// TIA Portal V17 export
// export: Created 2022-08-15T12:48:21.8497446Z, ExportSetting WithDefaults, DisplayName Totally Integrated Automation Portal, DisplayVersion V17, DisplayName TIA Portal Openness, DisplayVersion V17, DisplayName TIA Portal Version Control Interface, DisplayVersion V17, DisplayName SINAMICS Startdrive Advanced, DisplayVersion V17 Update1, DisplayName SINAMICS Startdrive G110M, G120, G120C, G120D, G120P, G115D, DisplayVersion V17 Update1, DisplayName SINAMICS Startdrive G130, G150, S120, S150, SINAMICS MV, S210, DisplayVersion V17 Update1, DisplayName STEP 7 Professional, DisplayVersion V17, DisplayName STEP 7 Safety, DisplayVersion V17, DisplayName WinCC Advanced, DisplayVersion V17
ORGANIZATION_BLOCK "Main"   // OB1, LAD, ProgramCycle
TITLE = "Main Program Sweep (Cycle)"
{ S7_Optimized_Access := 'TRUE' }
VERSION : 0.1
// stored: AutoNumber true, IsIECCheckEnabled false, SetENOAutomatically false
   VAR_INPUT
      Initial_Call : Bool;   // Initial call of this OB
      Remanence : Bool;   // =True, if remanent data are available
   END_VAR
BEGIN

REGION Network 1
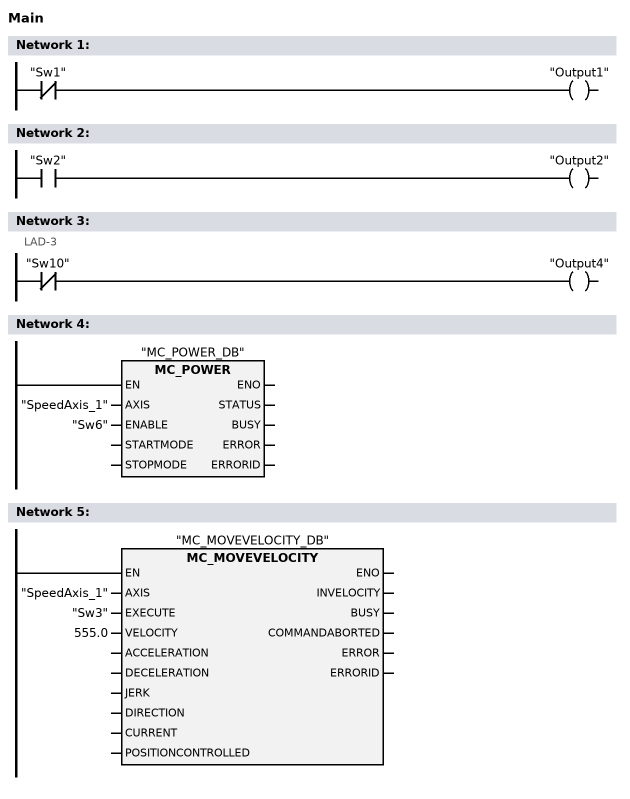
   RUNG wire#powerrail
      I_Contact( "Sw1" )
      Coil( "Output1" )
   END_RUNG
   // the same network as SCL:
   "Output1" := NOT "Sw1";
END_REGION

REGION Network 2
   RUNG wire#powerrail
      Contact( "Sw2" )
      Coil( "Output2" )
   END_RUNG
   // the same network as SCL:
   "Output2" := "Sw2";
END_REGION

REGION Network 3
   // LAD-3
   RUNG wire#powerrail
      I_Contact( "Sw10" )
      Coil( "Output4" )
   END_RUNG
   // the same network as SCL:
   "Output4" := NOT "Sw10";
END_REGION

REGION Network 4
   RUNG wire#powerrail
      "MC_POWER_DB".MC_POWER(Axis := "SpeedAxis_1", Enable := "Sw6", StartMode :=, StopMode :=, Status =>, Busy =>, Error =>, ErrorId =>)
   END_RUNG
   // the same network as SCL:
   "MC_POWER_DB"(Axis := "SpeedAxis_1", Enable := "Sw6");   // MC_POWER
END_REGION

REGION Network 5
   RUNG wire#powerrail
      "MC_MOVEVELOCITY_DB".MC_MOVEVELOCITY(Axis := "SpeedAxis_1", Execute := "Sw3", Velocity := 555.0, Acceleration :=, Deceleration :=, Jerk :=, Direction :=, Current :=, PositionControlled :=, InVelocity =>, Busy =>, CommandAborted =>, Error =>, ErrorId =>)
   END_RUNG
   // the same network as SCL:
   "MC_MOVEVELOCITY_DB"(Axis := "SpeedAxis_1", Execute := "Sw3", Velocity := 555.0);   // MC_MOVEVELOCITY
END_REGION
END_ORGANIZATION_BLOCK
